(* IEC 61131-3 sources: Lasal/CPU_5344_V01/Class/_Screen, 1 file *)

(* ---- _Screen.st ---- *)
(*!
<Class
	Name               = "_Screen"
	Revision           = "0.3"
	RealtimeTask       = "false"
	CyclicTask         = "false"
	BackgroundTask     = "false"
	Sigmatek           = "true"
	OSInterface        = "false"
	HighPriority       = "false"
	Automatic          = "false"
	UpdateMode         = "Prescan"
	IconPath           = ".\Class\_Screen\Screen.ico"
	SharedCommandTable = "true"
	Objectsize         = "(284,120)"
	Comment            = "userinterface">
	<Channels>
		<Server Name="Screen" Visualized="true" Initialize="false" WriteProtected="false" Retentive="false"/>
		<Client Name="ImA" Required="true" Internal="false"/>
		<Client Name="Lse" Required="true" Internal="false"/>
		<Client Name="No" Required="true" Internal="false"/>
	</Channels>
	<RevDoku>
		<Owner Company="sigmatek" Author="kolott"/>
		<Dokumentation Revision="0.3" Date="2016-11-07" Author="kolott" Company="sigmatek" Description="new virtual method S_WindowMoveable() is added"/>
		<Dokumentation Revision="0.2" Date="2013-02-28" Author="kolott" Company="sigmatek" Description="new methode S_CreateNew()&#13;&#10;icon added"/>
		<Dokumentation Revision="0.1" Date="2012-05-15" Author="kolott" Company="sigmatek" Description="optimization"/>
	</RevDoku>
</Class>
*)
_Screen : CLASS
  //Servers:
	Screen 	: SvrChCmd_DINT;
  //Clients:
	Lse 	: CltChCmd__Lse;
	No 	: CltCh_UDINT;
	ImA 	: CltCh_UDINT;
  //Variables:
		WhoAmI 	: _WHOAMI;
		FirstTime 	: BOOL;
  //Functions:

	FUNCTION _Screen
		VAR_OUTPUT
			ret_code 	: ConfStates;
		END_VAR;

	FUNCTION VIRTUAL GLOBAL Init;

	FUNCTION VIRTUAL GLOBAL S_End
		VAR_INPUT
			pic 	: ^void;
		END_VAR;

	FUNCTION VIRTUAL GLOBAL S_Run
		VAR_INPUT
			pic 	: ^void;
			event 	: ^_EVENT;
		END_VAR;

	FUNCTION VIRTUAL GLOBAL S_Ready
		VAR_INPUT
			pic 	: ^void;
			firsttime 	: BOOL;
		END_VAR;

	FUNCTION VIRTUAL GLOBAL S_Start
		VAR_INPUT
			pic 	: ^void;
			firsttime 	: BOOL;
		END_VAR;
				//! <Function Comment="method is used to create screen/window by program (without lse)&#13;&#10;kernel will call method only if screen/window is not present in lse-project" Name="S_CreateNew"/>
	FUNCTION VIRTUAL GLOBAL S_CreateNew
		VAR_INPUT
			psetup 	: ^_NEWSCREENPROP;
		END_VAR
		VAR_OUTPUT
			retcode 	: BOOL;
		END_VAR;
				//! <Function Comment="method is called to get information if window is moveable by user.&#13;&#10;return &apos;true&apos; if window is moveable, on the other hand &apos;false&apos;" Name="S_WindowMoveable"/>
	FUNCTION VIRTUAL GLOBAL S_WindowMoveable
		VAR_OUTPUT
			retcode 	: BOOL;
		END_VAR;
  //Tables:
	FUNCTION @STD
		VAR_OUTPUT
			ret_code	: CONFSTATES;
		END_VAR;
	FUNCTION GLOBAL TAB @CT_;
END_CLASS;

#pragma usingLtd _Lse

#pragma warning (disable : 73)

FUNCTION  _Screen::_Screen
VAR_OUTPUT
	ret_code		: CONFSTATES;
END_VAR

  FirstTime := TRUE;
  ret_code	:= C_OK;

END_FUNCTION

FUNCTION VIRTUAL GLOBAL _Screen::Init

  if(FirstTime = TRUE) then
    init_WHOAMI(#WhoAmI);
    WhoAmI.ima := (ImA.Read())$_IMA; //IMA_PICTURE;
    WhoAmI.no  := No.Read(); //0;
    Lse.AddScreen(this, #whoami);
    FirstTime := FALSE;
  end_if;

END_FUNCTION

FUNCTION VIRTUAL GLOBAL _Screen::S_Start
VAR_INPUT
	pic		    : ^VOID;
	firsttime	: BOOL;
END_VAR

END_FUNCTION

FUNCTION VIRTUAL GLOBAL _Screen::S_Ready
VAR_INPUT
	pic		    : ^VOID;
	firsttime	: BOOL;
END_VAR

END_FUNCTION

FUNCTION VIRTUAL GLOBAL _Screen::S_Run
VAR_INPUT
	pic		    : ^VOID;
	event		: ^_EVENT;
END_VAR

END_FUNCTION

FUNCTION VIRTUAL GLOBAL _Screen::S_End
VAR_INPUT
	pic		    : ^VOID;
END_VAR

END_FUNCTION

FUNCTION VIRTUAL GLOBAL _Screen::S_CreateNew
	VAR_INPUT
		psetup 	: ^_NEWSCREENPROP;
	END_VAR
	VAR_OUTPUT
		retcode 	: BOOL;
	END_VAR

  retcode := false;

END_FUNCTION

FUNCTION VIRTUAL GLOBAL _Screen::S_WindowMoveable
	VAR_OUTPUT
		retcode 	: BOOL;
	END_VAR

  retcode := true;

END_FUNCTION
